// TwinCAT 3 PLC project OEF_3
// ProgramVersion: 3.1.4024.0
// libraries:
//   Tc2_BABasic, * (Beckhoff Automation GmbH)
//   Tc2_Standard, * (Beckhoff Automation GmbH)
//   Tc2_System, * (Beckhoff Automation GmbH)
//   Tc3_Module, * (Beckhoff Automation GmbH)
//   VisuDialogs, * (System)
// project tree:
//   / GlobalTextList.TcGTLO, PlcTask.TcTTO, Visualization Manager.TcVMO (not stored)
//   POUs/ MAIN.TcPOU
//   VISUs/ Visualization.TcVIS
// (motion and I/O tree: see PLC project oef_1)
// real-time tasks:
//   TASK PlcTask: cycle T#10ms, priority 20, ADS port 350
//   TASK PlcTask1: cycle T#10ms, priority 21, ADS port 351
//   TASK PlcTask2: cycle T#10ms, priority 22, ADS port 352
//   TASK PlcTask3: cycle T#10ms, priority 23, ADS port 353
//   TASK PlcTask4: cycle T#10ms, priority 24, ADS port 354
// variable links:

CONFIGURATION OEF_3
    RESOURCE PLC ON TwinCAT3
        TASK PlcTask(INTERVAL := T#10ms, PRIORITY := 22);
        PROGRAM MAIN WITH PlcTask : MAIN;
    END_RESOURCE
END_CONFIGURATION

// ---- POUs/MAIN.TcPOU
PROGRAM MAIN
VAR
	Apotentiometer AT %I*: INT := 0;
	Npotentiometer AT %I*: INT;
	NScale AT %I*: INT := 100;
END_VAR

Apotentiometer := LREAL_TO_INT (F_Scale(Npotentiometer, 0,32767,0,NScale));

END_PROGRAM

// ---- GlobalTextList.TcGTLO
TEXTLIST GlobalTextList
  69 = 'de MAX waarde is'
  650 = 'de MAX waarde is %d'
  104 = 'de MAX waarde is %I'
  850 = 'Output value %i'
END_TEXTLIST

// ---- VISUs/Visualization.TcVIS
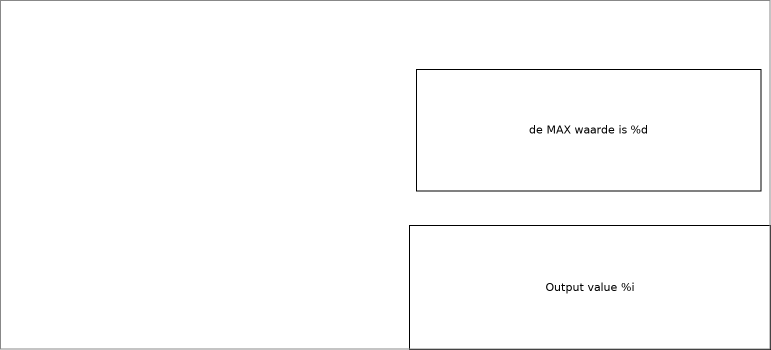
VISUALIZATION Visualization  // 771x350
    Rectangle (416,69 345x122), "de MAX waarde is %d", text variable: MAIN.NScale
        OnMouseClick: write the text variable via Default
    Rectangle (409,225 362x125), "Output value %i", text variable: MAIN.Apotentiometer
END_VISUALIZATION
